Staubli VAL3: setTrajItem.pgx

public program setTrajItem(TrajectoryItem& x_tTraj[], num x_nIndex)
begin
  //
  // set all the field
  //
  jEditPoint.tData[x_nIndex].tSuper=x_tTraj
  // active the save data
  bToSave=true
end
